{attribute 'linkalways'} 
{attribute 'no_explicit_call' := 'This FB is a CLASS and must be accessed using methods or properties'}
{attribute 'enable_dynamic_creation'}
FUNCTION_BLOCK FINAL OR_BOOL EXTENDS Node
VAR
	in1 : _BOOL(FALSE);
	in2 : _BOOL(FALSE);
	out : _BOOL(FALSE);
END_VAR

METHOD PUBLIC Clone : I_Node
VAR
	pNode : POINTER TO OR_BOOL;
END_VAR
pNode := __NEW(OR_BOOL);
Clone := pNode^;
END_METHOD

METHOD FB_init : BOOL
VAR_INPUT
	bInitRetains : BOOL; // if TRUE, the retain variables are initialized (warm start / cold start)
	bInCopyCode : BOOL;  // if TRUE, the instance afterwards gets moved into the copy code (online change)
END_VAR
AddInput('in1',THIS^.in1);
AddInput('in2',THIS^.in2);
AddOutput('out', THIS^.out);
END_METHOD

METHOD PROTECTED OnExecute
VAR
END_VAR
out.Value := in1.Value OR in2.Value;
END_METHOD

END_FUNCTION_BLOCK

(* stored: Version 1.1.0.1, ProductVersion 3.1.4024.15
   POU OR_BOOL: Id {1e8aeb72-6581-4aa4-ad4c-fc7bdc569f49}, SpecialFunc None
   Folder Constructor: Id {88cf18d5-fc27-4553-8168-604150687404}
   Method Clone: Id {e1b744f7-0250-4379-9ce3-99fac03a0f30}
   Method FB_init: Id {cf0984d6-3ce1-4ba0-8e57-a6552a8d4168}
   Method OnExecute: Id {52079313-4479-40c6-9005-6a6fc587dac9} *)
